(* PLC project  *)

CONFIGURATION StepIM_C
END_CONFIGURATION
